TYPE ST_XBox_Single_Directional_Joystick_NC_Options :
STRUCT
	// Inverts the direction of the axis
	bInverted : BOOL := FALSE;
	// Maximum Feedrate
	fMaxOverride : LREAL := 100.0;
	// Struct of parameters for MC_Halt command
	stXBox_NC_Halt_Dynamics : ST_XBox_NC_Halt_Dynamics;
END_STRUCT
END_TYPE

(* stored: Version 1.1.0.1, ProductVersion 3.1.4024.11
   DUT ST_XBox_Single_Directional_Joystick_NC_Options: Id {9bb20b1e-a972-4f2d-b27c-9cb410076cf4} *)
